FUNCTION_BLOCK FB_ADD_INT (* INT Addition *)
  (* Standard: 61499-1-D.1; Classification: Math *)
  (* Version 0.1, 2001-08-03, JHC, Rockwell Automation, Simplified version *)
  (* Version 0.0, 1998-04-15, JHC, Rockwell Automation, Original version *)
  (* Compiler header: package fb.rt.math; *)
  (* Compiler classdef: class FB_ADD_INT extends FBFunction2 *)
  (* Compiler Java IBM VisualAge 3.0 *)
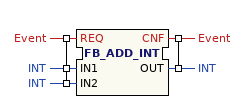
  EVENT_INPUT
    REQ WITH IN1, IN2;
  END_EVENT
  EVENT_OUTPUT
    CNF WITH OUT;
  END_EVENT
  VAR_INPUT
    IN1 : INT; (* Augend *)
    IN2 : INT; (* Addend *)
  END_VAR
  VAR_OUTPUT
    OUT : INT; (* Sum *)
  END_VAR
END_FUNCTION_BLOCK
